TYPE ST_MCHMIPrepareScreen_03_XX :
STRUCT
	btmpValue_03_XX	: BOOL;
END_STRUCT
END_TYPE

(* stored: Version 1.1.0.1
   DUT ST_MCHMIPrepareScreen_03_XX: Id {e5701d8d-c3b1-0fa2-16c8-dd973d024494} *)
